FUNCTION_BLOCK Hysteresis (* Analog to Digital with Hysteresis *)
  (* Standard: 61499-2 *)
  (* Version 1.0, 2026-05-08, 4diac IDE *)
  PACKAGE logiBUS::signalprocessing;
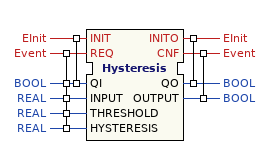
  EVENT_INPUT
    INIT : EInit WITH QI; (* Initialization Request *)
    REQ WITH QI, INPUT, THRESHOLD, HYSTERESIS; (* Normal Execution Request *)
  END_EVENT
  EVENT_OUTPUT
    INITO : EInit WITH QO; (* Initialization Confirm *)
    CNF WITH OUTPUT; (* Execution Confirmation *)
  END_EVENT
  VAR_INPUT
    QI : BOOL; (* Input event qualifier *)
    INPUT : REAL; (* Input value *)
    THRESHOLD : REAL := 0.0; (* Switch-off threshold *)
    HYSTERESIS : REAL := 0.1; (* Hysteresis band *)
  END_VAR
  VAR_OUTPUT
    QO : BOOL;
    OUTPUT : BOOL; (* Hysteresis output *)
  END_VAR
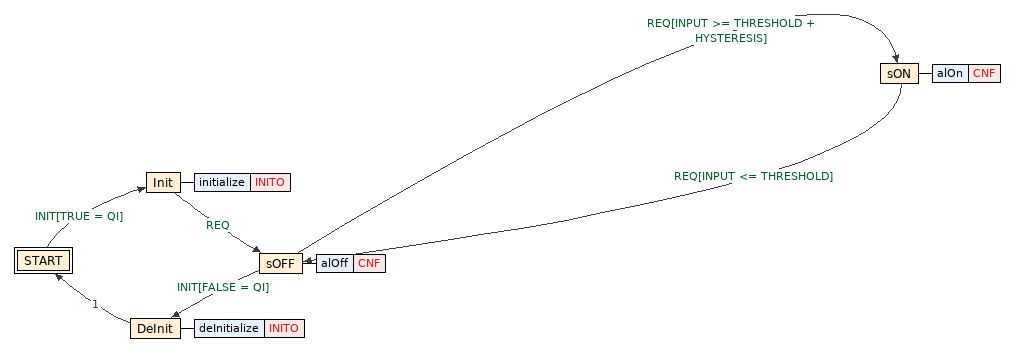
  EC_STATES
    START; (* Initial State *)
    Init : initialize -> INITO; (* Initialization *)
    sOFF : alOff -> CNF;
    DeInit : deInitialize -> INITO;
    sON : alOn -> CNF;
  END_STATES
  EC_TRANSITIONS
    START TO Init := INIT[TRUE = QI];
    Init TO sOFF := REQ;
    sOFF TO DeInit := INIT[FALSE = QI];
    sOFF TO sON := REQ[INPUT >= THRESHOLD + HYSTERESIS];
    DeInit TO START := 1;
    sON TO sOFF := REQ[INPUT <= THRESHOLD];
  END_TRANSITIONS
  ALGORITHM initialize IN ST:
QO := QI;
OUTPUT := BOOL#FALSE;
  END_ALGORITHM
  ALGORITHM deInitialize IN ST:
QO := BOOL#FALSE;
OUTPUT := BOOL#FALSE;
  END_ALGORITHM
  ALGORITHM alOff IN ST:
QO := QI;
OUTPUT := BOOL#FALSE;
  END_ALGORITHM
  ALGORITHM alOn IN ST:
QO := QI;
IF TRUE = QI THEN
	OUTPUT := BOOL#TRUE;
END_IF;
  END_ALGORITHM
END_FUNCTION_BLOCK
